KUKA KRL program: MASTER_125.src, MASTER_125.dat

--- MASTER_125.src ---
&ACCESS RVP
&REL 8
&PARAM EDITMASK = *
&PARAM TEMPLATE = C:\KRC\Roboter\Template\vorgabe
&PARAM DISKPATH = KRC:\R1\Program\Principal
DEF MASTER_125( )
;FOLD INI;%{PE}
  ;FOLD BASISTECH INI
    GLOBAL INTERRUPT DECL 3 WHEN $STOPMESS==TRUE DO IR_STOPM ( )
    INTERRUPT ON 3
    BAS (#INITMOV,0 )
  ;ENDFOLD (BASISTECH INI)
  ;FOLD USER INI
    ;Make your modifications here

  ;ENDFOLD (USER INI)
;ENDFOLD (INI)

;=======================================;
;       Cinética Automação/IFA          ;
;        Principal Master 125           ;
;                                       ;
;=======================================;

;FOLD Principal Master
$LOOP_MSG[] ="    ======Principal Master 125============="



;ENDFOLD (Principal Master)


 ;=======================================
  WHILE (NOT Fim_De_Trabalho)
   LOOP

     IF (Lib_Mesa_B) THEN
      LADO_B_OPERADOR()
     ENDIF

    IF (Lib_Soldar_Mesa_A) THEN

    NEW_MASTER_MESA_A()
   ENDIF
;=======================================

 IF (Lib_Mesa_A) THEN
   LADO_A_OPERADOR()
ENDIF


 IF (Lib_Soldar_Mesa_B) THEN

 MASTER_125_LADO_B()
   ENDIF

;=======================================
ENDLOOP

ENDWHILE
END

--- MASTER_125.dat ---
&ACCESS RVP
&REL 8
&PARAM EDITMASK = *
&PARAM TEMPLATE = C:\KRC\Roboter\Template\vorgabe
&PARAM DISKPATH = KRC:\R1\Program\Principal
DEFDAT  MASTER_125
;FOLD EXTERNAL DECLARATIONS;%{PE}%MKUKATPBASIS,%CEXT,%VCOMMON,%P
;FOLD BASISTECH EXT;%{PE}%MKUKATPBASIS,%CEXT,%VEXT,%P
EXT  BAS (BAS_COMMAND  :IN,REAL  :IN )
DECL INT SUCCESS
;ENDFOLD (BASISTECH EXT)
;FOLD USER EXT;%{E}%MKUKATPUSER,%CEXT,%VEXT,%P
;Make your modifications here

;ENDFOLD (USER EXT)
;ENDFOLD (EXTERNAL DECLARATIONS)
DECL BASIS_SUGG_T LAST_BASIS={POINT1[] "P0                      ",POINT2[] "P0                      ",CP_PARAMS[] "CPDAT0                  ",PTP_PARAMS[] "PDAT0                   ",CONT[] "                        ",CP_VEL[] "2.0                     ",PTP_VEL[] " 100                    ",SYNC_PARAMS[] "SYNCDAT                 ",SPL_NAME[] "S0                      ",A_PARAMS[] "ADAT0                   "}
ENDDAT
